// TIA Portal V19 export
TYPE "LEXCHANGETRAY_typeScanner_result"
// stored: Access Published
   STRUCT
      srCode { ExternalAccessible := 'False'; ExternalVisible := 'False'; ExternalWritable := 'False'} : String;
      traySize : Int := 24;
      ngOK : Int;
      ngSum : Int;
   END_STRUCT;
END_TYPE
